// TIA Portal V17 export
// export: Created 2026-08-04T13:46:49.5286309Z, ExportSetting WithDefaults, DisplayName Totally Integrated Automation Portal, DisplayVersion V17, DisplayName TIA Portal Openness, DisplayVersion V17, DisplayName TIA Portal Version Control Interface, DisplayVersion V17, DisplayName SINAMICS Startdrive Advanced, DisplayVersion V17, DisplayName SINAMICS Startdrive G130, G150, S120, S150, SINAMICS MV, G220, S200, S210, DisplayVersion V17, DisplayName SINAMICS Startdrive G110M, G120, G120C, G120D, G120P, G115D, DisplayVersion V17, DisplayName STEP 7 Professional, DisplayVersion V17, DisplayName STEP 7 Safety, DisplayVersion V17, DisplayName WinCC Basic/Comfort/Advanced, DisplayVersion V17, DisplayName WinCC Unified, DisplayVersion V17
ORGANIZATION_BLOCK "Cyclic interrupt"   // OB30, LAD, CyclicInterrupt
{ S7_Optimized_Access := 'TRUE' }
VERSION : 0.1
// stored: AutoNumber true, IsIECCheckEnabled false, SetENOAutomatically false
   VAR_INPUT
      Initial_Call : Bool;
      Event_Count : Int;
   END_VAR
   VAR_TEMP
      hscDATA : HW_HSC;
      temp : Real;
      reset_fault_simulation : Bool;
   END_VAR
BEGIN

REGION Network 1: Disable PWM
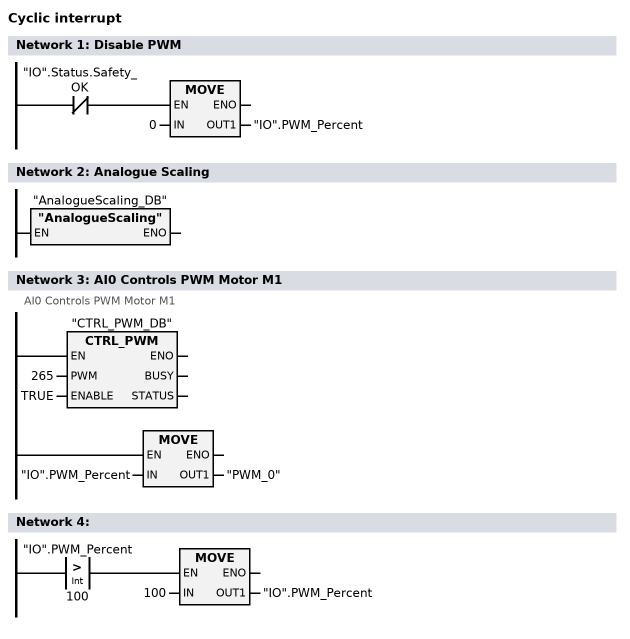
   RUNG wire#powerrail
      I_Contact( "IO".Status.Safety_OK )
      Move(in := 0, out1 => "IO".PWM_Percent)
   END_RUNG
   // the same network as SCL:
   IF NOT "IO".Status.Safety_OK THEN "IO".PWM_Percent := 0; END_IF;
END_REGION

REGION Network 2: Analogue Scaling
   RUNG wire#powerrail
      "AnalogueScaling_DB"()
   END_RUNG
   // the same network as SCL:
   "AnalogueScaling_DB"();   // "AnalogueScaling"
END_REGION

REGION Network 3: AI0 Controls PWM Motor M1
   // AI0 Controls PWM Motor M1
   RUNG wire#powerrail
      "CTRL_PWM_DB".CTRL_PWM(PWM := 265, ENABLE := TRUE, BUSY =>, STATUS =>)
   END_RUNG
   RUNG wire#powerrail
      Move(in := "IO".PWM_Percent, out1 => "PWM_0")
   END_RUNG
   // the same network as SCL:
   "CTRL_PWM_DB"(PWM := 265, ENABLE := TRUE);   // CTRL_PWM
   "PWM_0" := "IO".PWM_Percent;
END_REGION

REGION Network 4
   RUNG wire#powerrail
      { S7_Templates := "SrcType := Int" } GT_Contact(in1 := "IO".PWM_Percent, in2 := 100)
      Move(in := 100, out1 => "IO".PWM_Percent)
   END_RUNG
   // the same network as SCL:
   IF "IO".PWM_Percent > 100 THEN "IO".PWM_Percent := 100; END_IF;
END_REGION
END_ORGANIZATION_BLOCK
